// TIA Portal V20 export
DATA_BLOCK "BK03"   // DB302
// stored: MemoryReserve 100
   VAR
      "X10-1 JR OUT P&P2 Z-AXIS LIMIT SENSOR(-)" : Bool;
      "X10-2 JR OUT P&P2 Z-AXIS HOME SENSOR" : Bool;
      "X12-1 JR OUT P&P2 Z-AXIS LIMT SENSOR(+)" : Bool;
      "X12-2 JR OUT P&P2 STACK DETECT SENSOR" : Bool;
      "X14-1 JR OUT P&P2 CLAMP OPEN" : Bool;
      "X14-2 JR OUT P&P2 CLAMP CLOSE" : Bool;
      "X16-1 OUT P&P GRIPPER 2ND OPEN/CLOSE PRESSURE SENSOR" : Bool;
      "X16-2 OUT P&P GRIPPER 2ND Z-AXIS SAFETY PIN LOADING SENSOR" : Bool;
   END_VAR
BEGIN
END_DATA_BLOCK
